# B&R Automation Studio project PID_Lab
Automation Studio 4.7.3.93 SP; technology packages: mapp 5.6.2, mappControl 5.6.0

## Configuration pp500

CPU 5PP5CP.US15-00, AutomationRuntime C4.72, Build 4.1.2, Safety 0.0, Vc V4.72.1

CPU 5PP5CP.US15-02, AutomationRuntime C4.72, Build 4.1.2, Vc V4.72.1

### Task classes (Cpu.sw)
```
Libraries: MpTemp, MpAlarmX, MpBase, astime, runtime
```

### Task classes (Cpu.sw)
```
Cyclic#4:
  AlarmCtrl <- Control.AlarmCtrl.prg
  RecipeCtrl <- Control.RecipeCtrl.prg
Cyclic#5:
  TempCtrl <- Control.TempCtrl.prg
Binaries: FWRules, udbdef, arsvcreg, TCData, arconfig, User, Role, Config, sysconf, iomap, asfw, ashwac, ashwd
Libraries: mptemp, sys_lib, mpbase, astime, asieccon, fileio, runtime, brsystem
```

### Hardware
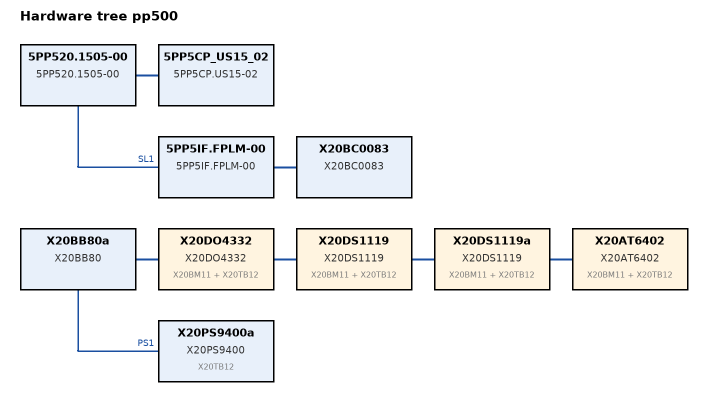
```
5PP520.1505-00 : 5PP520.1505-00 v2.0.3.1
  Connector IF3:
    ActivateDevice = 1
    Mode = Manual
    InternetAddress = 169.254.188.1
    SubnetMask = 255.255.0.0
  VcObjectName = Visu
5PP5CP_US15_02 : 5PP5CP.US15-02 v2.0.6.0  [SY -> 5PP520.1505-00.SY1]
  ConfigurationID = PID_Lab_pp500
  UserPartitionSize = 100
  RemMemDevice = PCI.1.PP5IF3.SRAM
  RemMemSize = 100
  RemanentGlobalPvSize = 50
  VolatileGlobalPvSize = 200000
  TimerDeviceType = EPLX2X
  TimerDevice = 5PP5IF.FPLM-00.IF1
  TaskClassIdleTime = 2000
  FileDevice1
  FileDeviceName1 = Recipes
  FileDevicePath1 = F:\Recipes
  FtpUser1
  FtpUsername1 = brcpu
  FtpUserPassword1 = rxMbsWslfkIXxy6fzmK6wAtRHG0v5cw0fRA9w62tUOs=
  FtpUserSalt1 = VKEEH50/
  FTPAccessRight1 = 0
  FTPdevice1 = ALL
5PP5IF.FPLM-00 : 5PP5IF.FPLM-00 v2.4.0.0  [SL -> 5PP520.1505-00.SL1]
X20AT6402 : X20AT6402 v1.0.6.0  [SS1 -> X20TB12d.SS; SL -> X20BM11c.SL1]
  Supervision = off
  DisableChannel05 = on
  DisableChannel06 = on
X20BB80a : X20BB80 v1.0.2.0
X20BC0083 : X20BC0083 v2.9.0.0  [PLK1 -> 5PP5IF.FPLM-00.IF1 [Cable Type=PowerlinkCable, Length=10, Version=1.0.0.2]; SL -> X20BB80a.SL1]
  Supervision = off
X20BM11 : X20BM11 v1.0.0.1  [X2X1 -> X20BB80a.IF1]
X20BM11a : X20BM11 v1.0.0.1  [X2X1 -> X20BM11.X2X2]
X20BM11b : X20BM11 v1.0.0.1  [X2X1 -> X20BM11a.X2X2]
X20BM11c : X20BM11 v1.0.0.1  [X2X1 -> X20BM11b.X2X2]
X20DO4332 : X20DO4332 v1.1.0.0  [SS1 -> X20TB12a.SS; SL -> X20BM11.SL1]
  Supervision = off
X20DS1119 : X20DS1119 v1.3.1.0  [SS1 -> X20TB12b.SS; SL -> X20BM11a.SL1]
  Supervision = off
  Channel01Config = outputPush
  Channel02Config = outputPush
  Channel03Config = outputPush
  DirectIOControlConfig = on
X20DS1119a : X20DS1119 v1.3.1.0  [SS1 -> X20TB12c.SS; SL -> X20BM11b.SL1]
  Supervision = off
  Channel01Config = outputPush
  DirectIOControlConfig = on
X20PS9400a : X20PS9400 v1.0.2.4  [SS1 -> X20TB12.SS; PS -> X20BB80a.PS1]
  Supervision = off
X20TB12 : X20TB12 v1.0.0.0
X20TB12a : X20TB12 v1.0.0.0
X20TB12b : X20TB12 v1.0.0.0
X20TB12c : X20TB12 v1.0.0.0
X20TB12d : X20TB12 v1.0.0.0
```

### Config_1.tempcontroller - 5PP5CP_US15_00/mappControl/Config_1.tempcontroller
```
Element gTempController_1 (Type=tempcontroller)
Element gTempController_2 (Type=tempcontroller)
Element gTempController_3 (Type=tempcontroller)
```

### Config_2.tempgroup - 5PP5CP_US15_00/mappControl/Config_2.tempgroup
```
Element gTempGroup_1 (Type=tempgroup)
  Linking:
    Subnodes:
      Zone[0] = gTempController_1
      Zone[1] = gTempController_2
      Zone[2] = gTempController_3
  Alarms = MpAlarmX
```

### IoMap.iom - 5PP5CP_US15_02/IoMap.iom
```iecst
VAR_CONFIG
	gDio.HeatOn[0] AT %QX."X20DO4332".DigitalOutput01;
	gDio.HeatOn[1] AT %QX."X20DO4332".DigitalOutput02;
	gDio.HeatOn[2] AT %QX."X20DO4332".DigitalOutput03;
	gDio.HeatOn[3] AT %QX."X20DO4332".DigitalOutput04;
	gDio.ZoneTemps[0] AT %IW."X20AT6402".Temperature01;
	gDio.ZoneTemps[1]  AT %IW."X20AT6402".Temperature02;
	gDio.ZoneTemps[2]  AT %IW."X20AT6402".Temperature03;
	gDio.ZoneTemps[3]  AT %IW."X20AT6402".Temperature04;
	gDio.ZoneFans[0] AT %QX."X20DS1119".DigitalOutput01;
	gDio.ZoneFans[1]  AT %QX."X20DS1119".DigitalOutput02;
	gDio.ZoneFans[2] AT %QX."X20DS1119".DigitalOutput03;
	gDio.DisturbanceFan AT %QX."X20DS1119a".DigitalOutput01;
END_VAR
```

### Config.tempcontroller - 5PP5CP_US15_02/mappControl/Config.tempcontroller
```
Element gTempController_1 (Type=tempcontroller)
  TempController:
    Type = 2
  Alarms = MpAlarmX
Element gTempController_2 (Type=tempcontroller)
  TempController:
    Type = 2
  Alarms = MpAlarmX
Element gTempController_3 (Type=tempcontroller)
  TempController:
    Type = 2
  Alarms = MpAlarmX
```

### Config_2.mpalarmxcore - 5PP5CP_US15_02/mappServices/Config_2.mpalarmxcore
```
Element gAlarmLink (Type=mpalarmxcore)
```

## Logical view

Binary libraries used (declarations not repeated): operator, runtime, astime, AsIecCon, MpAlarmX 5.06.2, MpBase 5.06.0, MpTemp 5.06.0, MpRecipe 5.06.2, sys_lib, MTTemp 2.01.0, MTTypes, brsystem

### Global.typ - Global data types
```iecst
TYPE
	MainState_enum :
		(
		MAIN_INIT := 0,
		MAIN_IDLE := 1,
		MAIN_HEAT := 2,
		MAIN_AUTOTUNE := 3,
		MAIN_ERROR := 4
		);
	RecipeCtrlState_enum :
		(
		RECIPE_INIT := 0,
		RECIPE_IDLE := 1,
		RECIPE_SAVE := 2,
		RECIPE_SAVE_AUTOTUNE := 3,
		RECIPE_LOAD := 4,
		RECIPE_DELETE := 5,
		RECIPE_ERROR := 6
		);
	TempCtrlState_enum :
		(
		TEMP_INIT := 0,
		TEMP_IDLE := 10,
		TEMP_ON := 20,
		TEMP_ON_MTZONE := 30,
		TEMP_AUTOTUNE := 40,
		TEMP_AUTOTUNE_ABORT := 41,
		TEMP_AUTOTUNE_MTZONE := 50,
		TEMP_ERROR := 60
		);
	MainCtrl_type : 	STRUCT
		Cmd : MainCmd_type;
		Status : MainStatus_type;
		Par : MainCtrlPar_type;
	END_STRUCT;
	MainCmd_type : 	STRUCT
		HeatOn : BOOL;
		AutotuneHeaters : BOOL;
		ErrorReset : BOOL;
		AutotuneMtHeater : BOOL;
		AbortTune : BOOL;
	END_STRUCT;
	MainStatus_type : 	STRUCT
		AutotuneDone : BOOL;
		AutotuneInProgress : BOOL;
	END_STRUCT;
	MainCtrlPar_type : 	STRUCT
		SingleZoneIndex : USINT;
	END_STRUCT;
	DIO_type : 	STRUCT
		ZoneTemps : ARRAY[0..3]OF INT;
		HeatOn : ARRAY[0..3]OF BOOL;
		ZoneFans : ARRAY[0..2]OF BOOL;
		DisturbanceFan : BOOL;
	END_STRUCT;
	Error_type : 	STRUCT
		ErrorActive : BOOL;
		ErrorSetID : UDINT;
		ErrorResetID : UDINT;
		ErrorName : STRING[100];
		LastState : MainState_enum;
		ErrorAcknowledgeID : UDINT;
	END_STRUCT;
	MainRecipeCtrl_type : 	STRUCT
		Par : RecipeParameters_type;
		Cmd : RecipeCmd_type;
		Status : RecipeStatus_type;
	END_STRUCT;
	RecipeParameters_type : 	STRUCT
		SelectedRecipeName : STRING[255];
		UISetup : MpRecipeUISetupType;
		UIConnect : MpRecipeUIConnectType;
		RecipeSaveIndex : USINT;
	END_STRUCT;
	RecipeCmd_type : 	STRUCT
		LoadRecipe : BOOL;
		SaveRecipe : BOOL;
		SaveAutotune : BOOL;
	END_STRUCT;
	RecipeStatus_type : 	STRUCT
		CommandDone : BOOL;
		SaveInProgress : BOOL;
		LoadInProgress : BOOL;
	END_STRUCT;
	TuneRecipe_type : 	STRUCT
		ControlTune : ARRAY[0..3]OF ControlTune_type;
		Update : BOOL;
	END_STRUCT;
	ControlTune_type : 	STRUCT
		PIDParameters : PIDParameterContainer_type;
		ProfileParameters : ProfileParametersContainer_type;
	END_STRUCT;
	PIDParameterContainer_type : 	STRUCT
		Heat : PIDParameter_type;
		Cool : PIDParameter_type;
	END_STRUCT;
	PIDParameter_type : 	STRUCT
		ProportionalGain : REAL;
		IntegrationTime : REAL;
		DerivativeTime : REAL;
		FilterTime : REAL;
	END_STRUCT;
	ProfileParametersContainer_type : 	STRUCT
		Heat : ProfileParameters_type;
		Cool : ProfileParameters_type;
	END_STRUCT;
	ProfileParameters_type : 	STRUCT
		SlewRate : REAL;
		FilterTime : REAL;
		DelayTime : REAL;
	END_STRUCT;
	TempInterface_type : 	STRUCT
		Trends : ARRAY[0..3]OF TempInterfaceTrends_type;
		Status : ARRAY[0..3]OF TempInterfaceStatus_type;
		PID : ARRAY[0..3]OF PIDParameterContainer_type;
		Enables : ARRAY[0..3]OF BOOL := [4(TRUE)];
	END_STRUCT;
	TempInterfaceTrends_type : 	STRUCT
		ActualTemp : REAL;
		SetTemp : REAL;
	END_STRUCT;
	TempInterfaceStatus_type : 	STRUCT
		TuningInProgress : BOOL;
		HeatOn : BOOL;
		FanOn : BOOL;
		ControlActive : BOOL;
	END_STRUCT;
	StateReporter_type : 	STRUCT
		Main : MainState_enum;
		Recipe : RecipeCtrlState_enum;
		Temp : TempCtrlState_enum;
	END_STRUCT;
END_TYPE
```

### Global.var - Global variables
```iecst
VAR CONSTANT
	TARGET_TEMP : USINT := 80;
	COOLDOWN_TEMP : USINT := 50;
END_VAR
VAR
	gAmbientTemperature : REAL := 28;
	gRecipeCtrl : MainRecipeCtrl_type;
	gMainState : MainState_enum := MAIN_INIT;
	gMainCtrl : MainCtrl_type;
END_VAR
VAR RETAIN
	gIndexOfLastLoadedTune : USINT := 0;
END_VAR
VAR
	gError : Error_type;
	gDio : DIO_type;
	gAlarmUIConnect : MpAlarmXListUIConnectType;
	gTempInterface : TempInterface_type;
	gTuneRecipe : TuneRecipe_type;
	gRecipeIO : TuneRecipe_type;
	gStateInfo : StateReporter_type;
END_VAR
```


### Program Logical/Control/MainCtrl (IEC)

#### Cyclic.st - Cyclic code
```iecst
(*********************************************************************************
 * Copyright:
 * Author:    TylerWoodley
 * Created:   August 2, 2020/3:50 PM
 *********************************************************************************)

PROGRAM _CYCLIC

	gStateInfo.Main := gMainState;

	IF NOT(gMainState = MAIN_INIT) THEN
		FOR index := 0 TO 2 DO
			 gTuneRecipe.ControlTune[index].PIDParameters := gTempInterface.PID[index];
		END_FOR;
	END_IF;

	CASE gMainState OF
		MAIN_INIT:
			gRecipeCtrl.Par.RecipeSaveIndex := gIndexOfLastLoadedTune;
			gRecipeCtrl.Cmd.LoadRecipe := TRUE;
			IF gRecipeCtrl.Status.CommandDone THEN
				gRecipeCtrl.Status.CommandDone := FALSE;
				gMainState := MAIN_IDLE;
			END_IF;
		MAIN_IDLE:
			IF gRecipeCtrl.Cmd.SaveAutotune THEN
				gMainState := MAIN_AUTOTUNE;
			END_IF
		MAIN_HEAT:
		MAIN_AUTOTUNE:
			IF gMainCtrl.Status.AutotuneDone THEN
				IF gRecipeCtrl.Status.CommandDone THEN
					gRecipeCtrl.Status.CommandDone      := FALSE;
					gMainCtrl.Status.AutotuneDone       := FALSE;
					gMainState := MAIN_IDLE;
				ELSE
					gMainCtrl.Status.AutotuneInProgress := FALSE;
					gRecipeCtrl.Cmd.SaveAutotune        := TRUE;
				END_IF
			ELSE
				gMainCtrl.Status.AutotuneInProgress     := TRUE;
			END_IF
		MAIN_ERROR:
	END_CASE;

END_PROGRAM
```

#### Variables.var - Local variables
```iecst
VAR
	i : UDINT;
	index : INT;
END_VAR
```

### Program Logical/Control/TempCtrl (IEC)

#### Cyclic.st - Cyclic code
```iecst
(*********************************************************************************
 * Copyright:
 * Author:    TylerWoodley
 * Created:   July 28, 2020/1:57 PM
 *********************************************************************************)

PROGRAM _CYCLIC

	gStateInfo.Temp := TempState;

	TempControllerFBs[ZONE_1_INDEX].MpLink := ADR(gTempController_1);
	TempControllerFBs[ZONE_2_INDEX].MpLink := ADR(gTempController_2);
	TempControllerFBs[ZONE_3_INDEX].MpLink := ADR(gTempController_3);

	TempGroup.Cmd.ErrorReset               := gMainCtrl.Cmd.ErrorReset;

	TempStatus.Error                       := TempGroup.MpZones[ZONE_1_INDEX].Out.Error OR
	                                          TempGroup.MpZones[ZONE_2_INDEX].Out.Error OR
	                                          TempGroup.MpZones[ZONE_3_INDEX].Out.Error;

	IF TempStatus.Error THEN
		IF TempStatus.TuningInProgress THEN
			TempState                      := TEMP_AUTOTUNE_ABORT;
		ELSE
			TempState                      := TEMP_ERROR;
		END_IF
	END_IF

	gMainCtrl.Status.AutotuneInProgress := TempStatus.TuningInProgress;

	FOR index := 0 TO 2 DO

		IF gTuneRecipe.Update THEN
			TempGroup.MpZones[index].In.Update := TRUE;
			UpdateControlParameters(gTuneRecipe.ControlTune[index], ADR(TempGroup.MpZones[index].In.Parameters));
		END_IF;

		TempStatus.CurrentTemp[index]                   := gDio.ZoneTemps[index] / 10;
		TempStatus.SetTemp[index]                       := TempGroup.MpZones[index].Out.Info.SetTemperature;
		TempStatus.HeatOn[index]                        := TempGroup.MpZones[index].Out.Heat;
		TempStatus.CoolOn[index]                        := TempGroup.MpZones[index].Out.Cool;

		TempGroup.MpZones[index].In.ActualTemperature   := TempStatus.CurrentTemp[index];
		TempStatus.AtTemp[index]                        := (TempGroup.MpZones[index].In.ActualTemperature = TARGET_TEMP);

		TempControllerFBs[index].Enable                 := gTempInterface.Enables[index];
		TempControllerFBs[index].ErrorReset             := TempGroup.Cmd.ErrorReset;
		TempControllerFBs[index].Parameters             := ADR(TempGroup.MpZones[index].In.Parameters);
		TempControllerFBs[index].Update                 := TempGroup.MpZones[index].In.Update;
		TempControllerFBs[index].SetTemperature         := TempGroup.MpZones[index].In.SetTemperature;
		TempControllerFBs[index].ActualTemperature      := TempGroup.MpZones[index].In.ActualTemperature;
		TempControllerFBs[index].Control                := TempGroup.MpZones[index].In.Control;
		TempControllerFBs[index].Tune                   := TempGroup.MpZones[index].In.Tune;

		TempGroup.MpZones[index].Out.Active             := TempControllerFBs[index].Active;
		TempGroup.MpZones[index].Out.ControlActive      := TempControllerFBs[index].ControlActive;
		TempGroup.MpZones[index].Out.Error              := TempControllerFBs[index].Error;
		TempGroup.MpZones[index].Out.Heat               := TempControllerFBs[index].Heat;
		TempGroup.MpZones[index].Out.Cool               := TempControllerFBs[index].Cool;
		TempGroup.MpZones[index].Out.Info               := TempControllerFBs[index].Info;
		TempGroup.MpZones[index].Out.StatusID           := TempControllerFBs[index].StatusID;
		TempGroup.MpZones[index].Out.UpdateDone         := TempControllerFBs[index].UpdateDone;
		TempGroup.MpZones[index].Out.TuningDone         := TempControllerFBs[index].TuningDone;

		gTempInterface.Status[index].ControlActive      := TempGroup.MpZones[index].Out.Active;
		gTempInterface.Status[index].FanOn              := TempGroup.MpZones[index].Out.Cool;
		gTempInterface.Status[index].HeatOn             := TempGroup.MpZones[index].Out.Heat;
		gTempInterface.Status[index].TuningInProgress   := TempGroup.MpZones[index].In.Tune;

		gTempInterface.Trends[index].ActualTemp         := TempStatus.CurrentTemp[index];
		gTempInterface.Trends[index].SetTemp            := TempStatus.SetTemp[index];
	END_FOR;

	IF gTuneRecipe.Update AND TempGroup.MpZones[ZONE_1_INDEX].Out.UpdateDone AND TempGroup.MpZones[ZONE_2_INDEX].Out.UpdateDone AND TempGroup.MpZones[ZONE_3_INDEX].Out.UpdateDone THEN
	  gTuneRecipe.Update := FALSE;
	END_IF;

	CASE TempState OF
		TEMP_INIT:
			TempState := TEMP_IDLE;
		TEMP_IDLE:
			IF gMainCtrl.Cmd.HeatOn THEN
				TempState                               := TEMP_ON;
			ELSIF gMainCtrl.Cmd.AutotuneHeaters THEN
				TempStatus.TuningInProgress         := TRUE;
				TempState                           := TEMP_AUTOTUNE;
			END_IF

		TEMP_ON:
			IF gMainCtrl.Cmd.HeatOn THEN
				FOR index := 0 TO 2 DO
					TempGroup.MpZones[index].In.SetTemperature := TARGET_TEMP;
					TempGroup.MpZones[index].In.Control        := TRUE;
					gDio.HeatOn[index]                         := TempGroup.MpZones[index].Out.Heat;
					gDio.ZoneFans[index]                       := TempGroup.MpZones[index].Out.Cool;
				END_FOR;
			ELSE
				FOR index := 0 TO 2 DO
					TempGroup.MpZones[index].In.Control        := FALSE;
					gDio.HeatOn[index]                         := FALSE;
					gDio.ZoneFans[index]                       := FALSE;
				END_FOR;

				TempState                                      := TEMP_IDLE;
			END_IF
		TEMP_AUTOTUNE:

			IF gMainCtrl.Cmd.AbortTune THEN
				TempState                                := TEMP_AUTOTUNE_ABORT;
			ELSE
				gMainCtrl.Cmd.AutotuneHeaters            := FALSE;

				IF TempStatus.TuningInProgress THEN

					FOR index := 0 TO 2 DO
						TempGroup.MpZones[index].In.Tune := TRUE;
						gDio.HeatOn[index]               := TempGroup.MpZones[index].Out.Heat;
						gDio.ZoneFans[index]             := TempGroup.MpZones[index].Out.Cool;
					END_FOR;
					TempStatus.TuningInProgress          := NOT (TempGroup.MpZones[0].Out.TuningDone AND
					                                             TempGroup.MpZones[1].Out.TuningDone AND
					                                             TempGroup.MpZones[2].Out.TuningDone);
				ELSE
					FOR index := 0 TO 2 DO
						TempGroup.MpZones[index].In.Tune := FALSE;
						gDio.HeatOn[index]               := FALSE;
						gDio.ZoneFans[index]             := FALSE;
					END_FOR;
					UpdateGlobalParameters(ADR(gTempInterface.Recipe), TempGroup);
					gMainCtrl.Status.AutotuneDone        := TRUE;
					TempState                            := TEMP_IDLE;
				END_IF;
			END_IF;

		TEMP_AUTOTUNE_ABORT:
			FOR index := 0 TO 2 DO
				TempGroup.MpZones[index].In.Tune := FALSE;
				gDio.HeatOn[index]               := FALSE;
				gDio.ZoneFans[index]             := FALSE;
			END_FOR;
			gMainCtrl.Status.AutotuneDone        := TRUE;

			IF TempStatus.Error THEN
				TempState                        := TEMP_ERROR;
			ELSE
				TempState                        := TEMP_IDLE;
			END_IF

		TEMP_ERROR:
			FOR index := 0 TO 2 DO
				TempGroup.MpZones[index].In.Tune     := FALSE;
			END_FOR;
			FOR index := 0 TO 3 DO
				gDio.HeatOn[index]                   := FALSE;
				gDio.ZoneFans[index]                 := FALSE;
			END_FOR;
			TempGroup.MtZone.Cmd.Abort               := TRUE;
			TempStatus.TuningInProgress              := FALSE;
			IF TempGroup.Cmd.ErrorReset THEN
				TempStatus.Error                     := FALSE;
				TempGroup.MtZone.Cmd.Abort           := FALSE;
				TempState                            := TEMP_IDLE;
			END_IF;
	END_CASE;

	TempControllerFBs[ZONE_1_INDEX]();
	TempControllerFBs[ZONE_2_INDEX]();
	TempControllerFBs[ZONE_3_INDEX]();
END_PROGRAM
```

#### Types.typ - Local data types
```iecst
TYPE
	TempStatus_type : 	STRUCT
		AmbientTemp : ARRAY[0..3]OF REAL;
		CurrentTemp : ARRAY[0..3]OF REAL;
		AtTemp : ARRAY[0..3]OF BOOL;
		TuningInProgress : BOOL;
		SetTemp : ARRAY[0..3]OF REAL;
		CoolOn : ARRAY[0..3]OF BOOL;
		HeatOn : ARRAY[0..3]OF BOOL;
		Error : BOOL;
	END_STRUCT;
	TempGroupCmd_type : 	STRUCT
		ErrorReset : BOOL;
	END_STRUCT;
	TempGroup_type : 	STRUCT
		MpZones : ARRAY[0..2]OF TempZone_type;
		MtZone : MtZone_Type;
		Cmd : TempGroupCmd_type;
	END_STRUCT;
	TempZone_type : 	STRUCT
		In : TempZoneInput_type;
		Out : TempZoneOutput_type;
	END_STRUCT;
	TempZoneInput_type : 	STRUCT
		Update : BOOL;
		SetTemperature : REAL;
		ActualTemperature : REAL;
		Control : BOOL;
		Parameters : MpTempControllerParType := (Tuning:=(Mode:=mpTEMP_TUNING_MODE_HEAT_COOL,SetPointHeat:=80,SetPointCool:=50));
		Tune : BOOL;
	END_STRUCT;
	TempZoneOutput_type : 	STRUCT
		Active : BOOL;
		Error : BOOL;
		StatusID : DINT;
		UpdateDone : BOOL;
		Heat : BOOL;
		Cool : BOOL;
		ControlActive : BOOL;
		Info : MpTempControllerInfoType;
		TuningDone : BOOL;
	END_STRUCT;
	MtZone_Type : 	STRUCT
		Profile : MtZoneProfile_type;
		Controller : MtZoneController_type;
		Tuning : MtZoneTuning_type;
		Cmd : MtZoneCmd_type;
		Status : MtZoneStatus_type;
	END_STRUCT;
	MtZoneStatus_type : 	STRUCT
		CurrentTemp : REAL;
	END_STRUCT;
	MtZoneController_type : 	STRUCT
		In : MtZoneControllerInput_type;
		Out : MtZoneControllerOutput_type;
	END_STRUCT;
	MtZoneControllerInput_type : 	STRUCT
		PIDParameters : MTTempControllerType;
		MaxHeatOut : REAL;
		MaxCoolOut : REAL;
		Update : BOOL;
		SetTemperature : REAL;
		ActTemperature : REAL;
		FeedForwardHeat : REAL;
		FeedForwardCool : REAL;
		ControlStatusIn : DINT;
		Enable : BOOL;
	END_STRUCT;
	MtZoneControllerOutput_type : 	STRUCT
		Active : BOOL;
		Error : BOOL;
		StatusID : DINT;
		UpdateDone : BOOL;
		HeatOut : REAL;
		CoolOut : REAL;
	END_STRUCT;
	MtZoneProfile_type : 	STRUCT
		In : MtZoneProfileInput_type;
		Out : MtZoneProfileOutput_type;
	END_STRUCT;
	MtZoneProfileInput_type : 	STRUCT
		PlantParameters : MTTempPlantType;
		MaxHeatOut : REAL;
		MaxCoolOut : REAL;
		Mode : MTTempProfileModeEnum;
		Update : BOOL;
		AmbientTemperature : REAL;
		SetPointTemperature : REAL;
		Start : BOOL;
		Abort : BOOL;
		InitTemperature : REAL;
		Init : BOOL;
	END_STRUCT;
	MtZoneProfileOutput_type : 	STRUCT
		Active : BOOL;
		Error : BOOL;
		StatusID : DINT;
		UpdateDone : BOOL;
		SetTemperature : REAL;
		FeedForwardHeat : REAL;
		FeedForwardCool : REAL;
		State : MTTempProfileStateEnum;
		InSetPoint : BOOL;
		InitDone : BOOL;
	END_STRUCT;
	MtZoneTuning_type : 	STRUCT
		In : MtZoneTuningInput_type;
		Out : MtZoneTuningOutput_type;
	END_STRUCT;
	MtZoneTuningInput_type : 	STRUCT
		AmbientTemperature : REAL;
		ActTemperature : REAL;
		HeatIn : REAL;
		CoolIn : REAL;
		Mode : MTTempTuningModeEnum;
		SetPointTemperature : REAL;
		CoolDownTemperature : REAL;
		StartSingleZone : BOOL;
		Abort : BOOL;
	END_STRUCT;
	MtZoneTuningOutput_type : 	STRUCT
		Active : BOOL;
		Error : BOOL;
		StatusID : DINT;
		SetTemperature : REAL;
		FeedForwardHeat : REAL;
		FeedForwardCool : REAL;
		TuningActive : BOOL;
		TuningDone : BOOL;
		State : MTTempTuningStateEnum;
		PIDParameters : MTTempControllerType;
		PIDParametersValid : BOOL;
		ControlStatusOut : DINT;
	END_STRUCT;
	MtZoneCmd_type : 	STRUCT
		Abort : BOOL;
	END_STRUCT;
END_TYPE
```

#### Variables.var - Local variables
```iecst
VAR
	TempGroup : TempGroup_type;
	index : USINT;
	TempControllerFBs : ARRAY[0..2] OF MpTempController;
	TempState : TempCtrlState_enum;
	TempStatus : TempStatus_type;
	MtTempControllerFB : MTTempController;
	MtTempProfileFB : MTTempProfile;
	MtTempTuningFB : MTTempTuning;
END_VAR
VAR CONSTANT
	ZONE_1_INDEX : USINT := 0;
	ZONE_2_INDEX : USINT := 1;
	ZONE_3_INDEX : USINT := 2;
	ZONE_4_INDEX : USINT := 3;
END_VAR
```

#### LocalFunctions.fun
```iecst
{REDUND_ERROR} FUNCTION UpdateControlParameters : BOOL (*Updates Control Parameters*) (*$GROUP=User,$CAT=User,$GROUPICON=User.png,$CATICON=User.png*)
	VAR_INPUT
		NewParValues : ControlTune_type;
		ControllerPar : REFERENCE TO MpTempControllerParType;
	END_VAR
END_FUNCTION

{REDUND_ERROR} FUNCTION UpdateGlobalParameters : BOOL (*Update Global Parameters from control info*) (*$GROUP=User,$CAT=User,$GROUPICON=User.png,$CATICON=User.png*)
	VAR_INPUT
		TuneRecipe : REFERENCE TO TuneRecipe_type;
		TempGroup : TempGroup_type;
	END_VAR
	VAR
		index : USINT;
	END_VAR
END_FUNCTION
```

#### UpdateControlParameters.st
```iecst
(*********************************************************************************
 * Copyright:
 * Author:    TylerWoodley
 * Created:   July 31, 2020/3:31 PM
 *********************************************************************************)

(* Updates Control Parameters *)
FUNCTION UpdateControlParameters

	ControllerPar.PID.Heat.DerivativeTime   := NewParValues.PIDParameters.Heat.DerivativeTime;
	ControllerPar.PID.Heat.FilterTime       := NewParValues.PIDParameters.Heat.FilterTime;
	ControllerPar.PID.Heat.IntegrationTime  := NewParValues.PIDParameters.Heat.IntegrationTime;
	ControllerPar.PID.Heat.ProportionalGain := NewParValues.PIDParameters.Heat.ProportionalGain;

	ControllerPar.PID.Cool.DerivativeTime   := NewParValues.PIDParameters.Cool.DerivativeTime;
	ControllerPar.PID.Cool.FilterTime       := NewParValues.PIDParameters.Cool.FilterTime;
	ControllerPar.PID.Cool.IntegrationTime  := NewParValues.PIDParameters.Cool.IntegrationTime;
	ControllerPar.PID.Cool.ProportionalGain := NewParValues.PIDParameters.Cool.ProportionalGain;

	ControllerPar.Profile.Heat.DelayTime    := NewParValues.ProfileParameters.Heat.DelayTime;
	ControllerPar.Profile.Heat.FilterTime   := NewParValues.ProfileParameters.Heat.FilterTime;
	ControllerPar.Profile.Heat.SlewRate     := NewParValues.ProfileParameters.Heat.SlewRate;

	ControllerPar.Profile.Heat.DelayTime    := NewParValues.ProfileParameters.Heat.DelayTime;
	ControllerPar.Profile.Heat.FilterTime   := NewParValues.ProfileParameters.Heat.FilterTime;
	ControllerPar.Profile.Heat.SlewRate     := NewParValues.ProfileParameters.Heat.SlewRate;

END_FUNCTION
```

#### UpdateGlobalParameters.st
```iecst
(*********************************************************************************
 * Copyright:
 * Author:    TylerWoodley
 * Created:   August 1, 2020/11:42 AM
 *********************************************************************************)

(* Update Global Parameters from control info *)
FUNCTION UpdateGlobalParameters

	FOR index := 0 TO 2 DO
		TuneRecipe.ControlTune[index].PIDParameters.Heat.DerivativeTime   := TempGroup.MpZones[index].Out.Info.Tuning.PIDParameters.Heat.DerivativeTime;
		TuneRecipe.ControlTune[index].PIDParameters.Heat.FilterTime       := TempGroup.MpZones[index].Out.Info.Tuning.PIDParameters.Heat.FilterTime;
		TuneRecipe.ControlTune[index].PIDParameters.Heat.IntegrationTime  := TempGroup.MpZones[index].Out.Info.Tuning.PIDParameters.Heat.IntegrationTime;
		TuneRecipe.ControlTune[index].PIDParameters.Heat.ProportionalGain := TempGroup.MpZones[index].Out.Info.Tuning.PIDParameters.Heat.ProportionalGain;

		TuneRecipe.ControlTune[index].PIDParameters.Cool.DerivativeTime   := TempGroup.MpZones[index].Out.Info.Tuning.PIDParameters.Cool.DerivativeTime;
		TuneRecipe.ControlTune[index].PIDParameters.Cool.FilterTime       := TempGroup.MpZones[index].Out.Info.Tuning.PIDParameters.Cool.FilterTime;
		TuneRecipe.ControlTune[index].PIDParameters.Cool.IntegrationTime  := TempGroup.MpZones[index].Out.Info.Tuning.PIDParameters.Cool.IntegrationTime;
		TuneRecipe.ControlTune[index].PIDParameters.Cool.ProportionalGain := TempGroup.MpZones[index].Out.Info.Tuning.PIDParameters.Cool.ProportionalGain;

		TuneRecipe.ControlTune[index].ProfileParameters.Heat.DelayTime    := TempGroup.MpZones[index].Out.Info.Tuning.ProfileParameters.Heat.DelayTime;
		TuneRecipe.ControlTune[index].ProfileParameters.Heat.FilterTime   := TempGroup.MpZones[index].Out.Info.Tuning.ProfileParameters.Heat.FilterTime;
		TuneRecipe.ControlTune[index].ProfileParameters.Heat.SlewRate     := TempGroup.MpZones[index].Out.Info.Tuning.ProfileParameters.Heat.SlewRate;

		TuneRecipe.ControlTune[index].ProfileParameters.Cool.DelayTime    := TempGroup.MpZones[index].Out.Info.Tuning.ProfileParameters.Cool.DelayTime;
		TuneRecipe.ControlTune[index].ProfileParameters.Cool.FilterTime   := TempGroup.MpZones[index].Out.Info.Tuning.ProfileParameters.Cool.FilterTime;
		TuneRecipe.ControlTune[index].ProfileParameters.Cool.SlewRate     := TempGroup.MpZones[index].Out.Info.Tuning.ProfileParameters.Cool.SlewRate;
	END_FOR;
	(*
	TuneRecipe.ControlTune[3].PIDParameters.Heat.DerivativeTime           := TempGroup.MtZone.Tuning.Out.PIDParameters.Heating.DerivativeTime;
	TuneRecipe.ControlTune[3].PIDParameters.Heat.FilterTime               := TempGroup.MtZone.Tuning.Out.PIDParameters.Heating.FilterTime;
	TuneRecipe.ControlTune[3].PIDParameters.Heat.IntegrationTime          := TempGroup.MtZone.Tuning.Out.PIDParameters.Heating.IntegrationTime;
	TuneRecipe.ControlTune[3].PIDParameters.Heat.ProportionalGain         := TempGroup.MtZone.Tuning.Out.PIDParameters.Heating.Gain;

	TuneRecipe.ControlTune[3].PIDParameters.Cool.DerivativeTime           := TempGroup.MtZone.Tuning.Out.PIDParameters.Cooling.DerivativeTime;
	TuneRecipe.ControlTune[3].PIDParameters.Cool.FilterTime               := TempGroup.MtZone.Tuning.Out.PIDParameters.Cooling.FilterTime;
	TuneRecipe.ControlTune[3].PIDParameters.Cool.IntegrationTime          := TempGroup.MtZone.Tuning.Out.PIDParameters.Cooling.IntegrationTime;
	TuneRecipe.ControlTune[3].PIDParameters.Cool.ProportionalGain         := TempGroup.MtZone.Tuning.Out.PIDParameters.Cooling.Gain;
	*)
END_FUNCTION
```

#### UpdateMtControlParameters.st - not listed in the package file held
```iecst
(*********************************************************************************
 * Copyright:
 * Author:    TylerWoodley
 * Created:   August 1, 2020/11:20 AM
 *********************************************************************************)

(* TODO: Add your comment here *)
FUNCTION UpdateMtControlParameters

	ControllerPar.Heating.DerivativeTime  := NewParValues.PIDParameters.Heat.DerivativeTime;
	ControllerPar.Heating.FilterTime      := NewParValues.PIDParameters.Heat.FilterTime;
	ControllerPar.Heating.IntegrationTime := NewParValues.PIDParameters.Heat.IntegrationTime;
	ControllerPar.Heating.Gain            := NewParValues.PIDParameters.Heat.ProportionalGain;

	ControllerPar.Cooling.DerivativeTime  := NewParValues.PIDParameters.Cool.DerivativeTime;
	ControllerPar.Cooling.FilterTime      := NewParValues.PIDParameters.Cool.FilterTime;
	ControllerPar.Cooling.IntegrationTime := NewParValues.PIDParameters.Cool.IntegrationTime;
	ControllerPar.Cooling.Gain            := NewParValues.PIDParameters.Cool.ProportionalGain;

END_FUNCTION
```

### Program Logical/Control/AlarmCtrl (IEC)

#### Variables.var
```iecst
VAR
	AlarmFB : MpAlarmXCore;
	AlarmUISetup : MpAlarmXListUISetupType;
	AlarmListUI : MpAlarmXListUI;
END_VAR
```

#### Cyclic.st
```iecst
(*********************************************************************************
 * Copyright:
 * Author:    TylerWoodley
 * Created:   July 29, 2020/8:34 PM
 *********************************************************************************)

PROGRAM _CYCLIC
	AlarmFB.MpLink := ADR(gAlarmLink);
	AlarmFB.Enable := TRUE;

	AlarmListUI.MpLink    := ADR(gAlarmLink);
	AlarmListUI.Enable    := TRUE;
	AlarmListUI.UISetup   := AlarmUISetup;
	AlarmListUI.UIConnect := ADR(gAlarmUIConnect);

	AlarmFB();
	AlarmListUI();

END_PROGRAM
```

### Program Logical/Control/RecipeCtrl (IEC)

#### Types.typ
```iecst
TYPE
	RecipeCtrl_type : 	STRUCT
		In : RecipeCtrlInput_type;
		Out : RecipeCtrlOutput_type;
		Par : RecipeCtrlPar_type;
	END_STRUCT;
	RecipeCtrlInput_type : 	STRUCT
		ErrorReset : BOOL;
		DeviceName : STRING[50];
		FileName : STRING[255];
		Save : BOOL;
		Load : BOOL;
	END_STRUCT;
	RecipeCtrlOutput_type : 	STRUCT
		Active : BOOL;
		Error : BOOL;
		StatusID : DINT;
		CommandDone : BOOL;
		Info : MpRecipeXmlInfoType;
	END_STRUCT;
	RecipeCtrlPar_type : 	STRUCT
		In : RecipeCtrlParInput_type;
		Out : RecipeCtrlParOutput_type;
	END_STRUCT;
	RecipeCtrlParInput_type : 	STRUCT
		ErrorReset : BOOL;
		PVName : STRING[100];
	END_STRUCT;
	RecipeCtrlParOutput_type : 	STRUCT
		Active : BOOL;
		Error : BOOL;
		StatusID : DINT;
		Info : MpRecipeInfoType;
	END_STRUCT;
END_TYPE
```

#### Variables.var
```iecst
VAR CONSTANT
	EMPTY_FILENAME : STRING[255] := '';
	PV_NAME : STRING[100] := 'gRecipeIO';
	AUTOTUNE_FILENAME_INDEX : USINT := 0;
	DEVICE_NAME : STRING[50] := 'Recipes';
END_VAR
VAR
	RecipeUIFB : MpRecipeUI;
	RecipeParFB : MpRecipeRegPar;
	RecipeCtrl : RecipeCtrl_type;
	RecipeXmlFB : MpRecipeXml;
	RecipeState : RecipeCtrlState_enum := RECIPE_INIT;
	RecipeNames : ARRAY[0..12] OF STRING[255] := ['Autotune.xml','Tune_01.xml','Tune_02.xml','Tune_03.xml','Tune_04.xml','Tune_05.xml','Tune_06.xml','Tune_07.xml','Tune_08.xml','Tune_09.xml','Tune_10.xml','Tune_11.xml','Tune_12.xml'];
	index : INT;
END_VAR
```

#### Cyclic.st
```iecst
(*********************************************************************************
 * Copyright:
 * Author:    TylerWoodley
 * Created:   July 29, 2020/10:21 PM
 *********************************************************************************)

PROGRAM _CYCLIC

	gStateInfo.Recipe                  := RecipeState;

	gRecipeCtrl.Par.SelectedRecipeName := RecipeNames[gRecipeCtrl.Par.RecipeSaveIndex];

	RecipeCtrl.In.DeviceName           := DEVICE_NAME;

	RecipeXmlFB.MpLink                 := ADR(gRecipeXml);
	RecipeXmlFB.Enable                 := TRUE;
	RecipeXmlFB.ErrorReset             := RecipeCtrl.In.ErrorReset;
	RecipeXmlFB.DeviceName             := ADR(DEVICE_NAME);
	RecipeXmlFB.FileName               := ADR(RecipeCtrl.In.FileName);
	RecipeXmlFB.Load                   := RecipeCtrl.In.Load;
	RecipeXmlFB.Save                   := RecipeCtrl.In.Save;

	RecipeParFB.MpLink                 := ADR(gRecipeXml);
	RecipeParFB.Enable                 := TRUE;
	RecipeParFB.ErrorReset             := RecipeCtrl.In.ErrorReset;
	RecipeParFB.PVName                 := ADR(PV_NAME);

	RecipeUIFB.MpLink                  := ADR(gRecipeXml);
	RecipeUIFB.Enable                  := TRUE;
	RecipeUIFB.ErrorReset              := RecipeCtrl.In.ErrorReset;
	RecipeUIFB.UIConnect               := ADR(gRecipeCtrl.Par.UIConnect);
	RecipeUIFB.UISetup                 := gRecipeCtrl.Par.UISetup;

	RecipeCtrl.Out.Active              := RecipeXmlFB.Active;
	RecipeCtrl.Out.Error               := RecipeXmlFB.Error;
	RecipeCtrl.Out.StatusID            := RecipeXmlFB.StatusID;
	RecipeCtrl.Out.CommandDone         := RecipeXmlFB.CommandDone;
	RecipeCtrl.Out.Info                := RecipeXmlFB.Info;

	RecipeCtrl.Par.Out.Active          := RecipeParFB.Active;
	RecipeCtrl.Par.Out.Error           := RecipeParFB.Error;
	RecipeCtrl.Par.Out.StatusID        := RecipeParFB.StatusID;
	RecipeCtrl.Par.Out.Info            := RecipeParFB.Info;

	IF RecipeCtrl.Out.Error OR RecipeCtrl.Par.Out.Error THEN
		RecipeState := RECIPE_ERROR;
	END_IF;

	CASE RecipeState OF
		RECIPE_INIT:
			RecipeState := RECIPE_IDLE;

		RECIPE_IDLE:
			IF gRecipeCtrl.Cmd.SaveRecipe THEN
				gRecipeCtrl.Cmd.SaveRecipe       := FALSE;
				RecipeState                      := RECIPE_SAVE;
			ELSIF gRecipeCtrl.Cmd.SaveAutotune THEN
				gRecipeCtrl.Cmd.SaveAutotune     := FALSE;
				gRecipeCtrl.Par.RecipeSaveIndex  := AUTOTUNE_FILENAME_INDEX;
				gRecipeCtrl.Cmd.SaveRecipe       := TRUE;
			ELSIF gRecipeCtrl.Cmd.LoadRecipe THEN
				gRecipeCtrl.Cmd.LoadRecipe       := FALSE;
				RecipeState                      := RECIPE_LOAD;
			END_IF;

		RECIPE_SAVE:
			IF NOT EDGEPOS(RecipeCtrl.Out.CommandDone) THEN
				gRecipeIO                         := gTuneRecipe;
				gRecipeCtrl.Status.CommandDone    := FALSE;
				gRecipeCtrl.Status.SaveInProgress := TRUE;
				RecipeCtrl.In.FileName            := gRecipeCtrl.Par.SelectedRecipeName;
				RecipeCtrl.In.Save                := TRUE;
			ELSE
				gRecipeCtrl.Status.CommandDone    := TRUE;
				gRecipeCtrl.Status.SaveInProgress := FALSE;
				RecipeCtrl.In.Save                := FALSE;
				RecipeCtrl.In.FileName            := EMPTY_FILENAME;
				RecipeState                       := RECIPE_IDLE;
			END_IF;

		RECIPE_LOAD:
			IF NOT EDGEPOS(RecipeCtrl.Out.CommandDone) THEN
				gRecipeCtrl.Status.CommandDone    := FALSE;
				gRecipeCtrl.Status.LoadInProgress := TRUE;
				RecipeCtrl.In.FileName            := gRecipeCtrl.Par.SelectedRecipeName;
				RecipeCtrl.In.Load                := TRUE;
			ELSE
				gTempInterface.Recipe             := gRecipeIO;
				gTempInterface.Recipe.Update             := TRUE;
				gRecipeCtrl.Status.CommandDone    := TRUE;
				gIndexOfLastLoadedTune            := gRecipeCtrl.Par.RecipeSaveIndex;
				gRecipeCtrl.Status.LoadInProgress := FALSE;
				RecipeCtrl.In.Load                := FALSE;
				RecipeCtrl.In.FileName            := EMPTY_FILENAME;
				RecipeState                       := RECIPE_IDLE;
			END_IF;

		RECIPE_DELETE:

		RECIPE_ERROR:
			RecipeCtrl.In.Load     := FALSE;
			RecipeCtrl.In.Save     := FALSE;
			RecipeCtrl.In.FileName := EMPTY_FILENAME;
			IF RecipeCtrl.In.ErrorReset THEN
	  			RecipeState        := RECIPE_IDLE;
			END_IF;

	END_CASE;

	RecipeXmlFB();
	RecipeParFB();
	//RecipeUIFB();

END_PROGRAM
```

- Visualisation Logical/Vis/Visu (not shown)

### Program Logical/Vis/VisCtrl (IEC)

#### Types.typ
```iecst
TYPE
	Vis_type : 	STRUCT
		Alarms : VisAlarms_type;
		Temp : TempInterface_type;
		States : StateReporter_type;
	END_STRUCT;
	VisAlarms_type : 	STRUCT
		AlarmListConnect : MpAlarmXListUIConnectType;
	END_STRUCT;
	Page_enum :
		(
		PAGE_START,
		PAGE_MAIN,
		PAGE_TREND,
		PAGE_ALARM,
		PAGE_ALARMHISTORY,
		PAGE_SETUP,
		PAGE_SDM
		);
END_TYPE
```

#### Variables.var
```iecst
VAR
	Vis : Vis_type;
	Page : Page_enum := PAGE_START;
	ChangePage : Page_enum := PAGE_START;
	index : INT;
END_VAR
```

#### Cyclic.st
```iecst
(*********************************************************************************
 * Copyright:
 * Author:    TylerWoodley
 * Created:   July 30, 2020/11:50 AM
 *********************************************************************************)

PROGRAM _CYCLIC
	FOR index := 0 TO 2 DO
		Vis.Temp.Trends[index] := gTempInterface.Trends[index];
		Vis.Temp.Status[index] := gTempInterface.Status[index];
	END_FOR;

	Vis.States := gStateInfo;

	IF (Page = PAGE_START) THEN

		IF EDGEPOS(gMainState = MAIN_IDLE) THEN
			ChangePage := PAGE_MAIN;
		END_IF;
	ELSE

	END_IF;

	IF EDGENEG(gRecipeCtrl.Status.LoadInProgress) THEN
		Vis.Temp.Recipe := gTuneRecipe;
	ELSE
		gTempInterface.Recipe := Vis.Temp.Recipe;
	END_IF

END_PROGRAM
```

Listed in the project but not available here: Logical/Control/MainCtrl/Init.st, Logical/Control/MainCtrl/Exit.st, Logical/Control/MainCtrl/Types.typ
